FUNCTION F_Error_Check : INT
VAR_INPUT
	ErrorCode															: DWORD;
	Error																: INT;
END_VAR
VAR
END_VAR

// F_Error_Check
// Rev 1.0 - October 9, 2024


F_Error_Check															:= SEL((ErrorCode AND LREAL_TO_DWORD(EXPT(2, Error))) > 0, 0, DWORD_TO_INT(ErrorCode));

END_FUNCTION

(* stored: Version 1.1.0.1, ProductVersion 3.1.4024.13
   POU F_Error_Check: Id {fbff525d-4e2f-4095-9d4a-02c0960437a2}, SpecialFunc None *)
